// TIA Portal V15.1 export
// export: Created 2024-05-17T05:38:11.0330835Z, ExportSetting WithDefaults, DisplayName Totally Integrated Automation Portal, DisplayVersion V15.1 Update 5, DisplayName TIA Portal Openness, DisplayVersion V15.1 Update 5, DisplayName SINAMICS Startdrive Advanced, DisplayVersion V15.1, DisplayName G130, G150, S120, S150, SINAMICS MV, S210, DisplayVersion V15.1, DisplayName G110M, G120, G120C, G120D, G120P, DisplayVersion V15.1, DisplayName STEP 7 Professional, DisplayVersion V15.1 Update 5, DisplayName STEP 7 Safety, DisplayVersion V15.1, DisplayName WinCC Professional, DisplayVersion V15.1 Update 5, DisplayName SIMATIC Visualization Architect, DisplayVersion V15.1
DATA_BLOCK "_DiagPLCOverview"   // DB251
{ S7_Optimized_Access := 'FALSE' }
AUTHOR : VCC
VERSION : 0.1
// stored: AutoNumber false, DBAccessibleFromOPCUA true, IsOnlyStoredInLoadMemory false, IsWriteProtectedInAS false
   VAR RETAIN
      "209000NCP01PNIODiag" { ExternalAccessible := 'False'; ExternalVisible := 'False'; ExternalWritable := 'False'} : "AlarmBits";   // PNIODiag Alarm Bits / Alarm A
      "209000NCP01Com" { ExternalAccessible := 'False'; ExternalVisible := 'False'; ExternalWritable := 'False'} : "AlarmBits";   // Com Alarm Bits
      DPComPLC212 { ExternalAccessible := 'False'; ExternalVisible := 'False'; ExternalWritable := 'False'} : "AlarmBits";   // DPCom PLC212 Alarm Bits / Alarm A
      PNComPLC308 { ExternalAccessible := 'False'; ExternalVisible := 'False'; ExternalWritable := 'False'} : "AlarmBits";   // PNCom PLC308 Alarm Bits / Alarm A
      AlarmA { ExternalAccessible := 'False'; ExternalVisible := 'False'; ExternalWritable := 'False'} : Bool;   // Alarm A
      AlarmB { ExternalAccessible := 'False'; ExternalVisible := 'False'; ExternalWritable := 'False'} : Bool;   // Alarm B
      AlarmC { ExternalAccessible := 'False'; ExternalVisible := 'False'; ExternalWritable := 'False'} : Bool;   // Alarm C
      AlarmD { ExternalAccessible := 'False'; ExternalVisible := 'False'; ExternalWritable := 'False'} : Bool;   // Alarm D
      AlarmABCondition : Bool;   // Alarm AB condition
      H_209000NCP01PNIODiagIAnim : Word;   // Icon Animation
      H_209000NCP01ComVDIAnim : Word;   // Icon Animation
      H_DPComPLC212IAnim : Word;   // Icon Animation
      H_PNComPLC308IAnim : Word;   // Icon Animation
      H_Anim : Word;   // Animation
      H_DBnr : Int;   // DB number
      H_HMICmd : Word;   // HMI Command
      Edge001 { ExternalAccessible := 'False'; ExternalVisible := 'False'; ExternalWritable := 'False'} : Bool;   // Edge
      Edge002 { ExternalAccessible := 'False'; ExternalVisible := 'False'; ExternalWritable := 'False'} : Bool;   // Edge
      TimerResetPNStatus { ExternalAccessible := 'False'; ExternalVisible := 'False'; ExternalWritable := 'False'} : TP_TIME;   // Timer
   END_VAR
BEGIN
END_DATA_BLOCK
